{attribute 'qualified_only'}
{attribute 'strict'}
TYPE ActiveWindowStateType :
(
	EXPERIMENT_WINDOW := 0,
	CALIBRATION_WINDOW := 1, 
	PARTICIPANT_WINDOW := 2
) SINT := EXPERIMENT_WINDOW;
END_TYPE

(* stored: Version 1.1.0.1, ProductVersion 3.1.4024.12
   DUT ActiveWindowStateType: Id {fc9328e0-26f3-41ff-8943-5bd343f7b707} *)
